# EPICS autosave request: support/ccd/1-10/iocBoot/iocMarCCD/auto_settings.req
file "ccd_settings.req", P=marCCD:, C=det1:
